// TIA Portal V20 export
DATA_BLOCK "HmiInterface"   // DB177
// stored: Access Published, MemoryReserve 100, Namespace Unit1.Em4
   VAR
      em : "LAF_typeEmInterface";
      cm : "Unit1.Em4.typeCmHmiInterface";
      sideTapeLoading : "LER_typeSequenceInterface";
      sideTapeAttachment : "LER_typeSequenceInterface";
      sideTapeFixStage : "LER_typeSequenceInterface";
      SideTapeIdleTime : "Unit1.Em4.typeSideTapeIdleTimeHmiInterface";
      sideTapeCuttingCount : "LER_typeAlarmCounterInterface";
      cmSideTapeSafetyPin : "LBC_typeDigitalSignalInterface";
      cmSideTapeJRDetect : "LBC_typeDigitalSignalInterface";
      cmSideTapeDiameter : "LBC_typeDigitalSignalInterface";
      cmSideTapeFixStageAxisX : "LBC_typeAxis64PosInterface";
      cmSideTapeFixStageAxisC : "LBC_typeAxis64PosInterface";
      cmSideTapeAttachmentAxisX : "LBC_typeAxis64PosInterface";
      cmSideTapeAttachmentAxisY : "LBC_typeAxis64PosInterface";
      cmSideTapeLoadingDownUp : "LBC_typeTwoWayActuatorInterface";
      cmSideTapeLoadingClampOpenClose : "LBC_typeTwoWayActuatorInterface";
      cmSideTapeCutterBwdFwd : "LBC_typeTwoWayActuatorInterface";
      cmSideTapeCutterClampBwdFwd : "LBC_typeTwoWayActuatorInterface";
      cmSideTapeTensionBwdFwd : "LBC_typeTwoWayActuatorInterface";
      cmSideTapeAttachmentLeftBwdFwd : "LBC_typeTwoWayActuatorInterface";
      cmSideTapeAttachmentRightBwdFwd : "LBC_typeTwoWayActuatorInterface";
      cmSideTapeAttachmentBtmBwdFwd : "LBC_typeTwoWayActuatorInterface";
      cmSideTapeFixStageClampOpenClose : "LBC_typeTwoWayActuatorInterface";
      cmSideTapeAttachment1TopVaccumOffOn : "LBC_typeTwoWayActuatorInterface";
      cmSideTapeAttachment1BtmVaccumOffOn : "LBC_typeTwoWayActuatorInterface";
      cmSideTapeAttachment2TopVaccumOffOn : "LBC_typeTwoWayActuatorInterface";
      cmSideTapeAttachment2BtmVaccumOffOn : "LBC_typeTwoWayActuatorInterface";
      cmQrHandyReader : "LER_typeDM8700Interface";
      "=====사용유무 확인필요=====" { ExternalAccessible := 'False'; ExternalVisible := 'False'; ExternalWritable := 'False'} : Bool;
      sequenceUnused : Array[0.._.U1EM4_NO_OF_SEQUENCE] of Bool;
      intCondition : "Unit1.Em4.typeIntConditionHmiInterface";
   END_VAR
BEGIN
   SideTapeIdleTime.processCount := T#5M;
   sideTapeCuttingCount.referenceDesignator := WSTRING#'Em4 Side Tape Cutting Count';
   sideTapeCuttingCount.ProcessValue.faultCount := 5000;
   sideTapeCuttingCount.SetValue.faultCount := 50000;
   cmSideTapeFixStageAxisC.configuration.setPositions[0]."name" := 'Wait [Tape1]';
   cmSideTapeFixStageAxisC.configuration.setPositions[1]."name" := 'Tape2';
   cmSideTapeFixStageAxisC.configuration.setPositions[2]."name" := 'Tape3';
   cmSideTapeFixStageAxisC.configuration.setPositions[3]."name" := 'Tape4';
   cmSideTapeAttachmentAxisX.configuration.setPositions[0]."name" := 'Wait';
   cmSideTapeAttachmentAxisX.configuration.setPositions[1]."name" := 'Right Tape Get';
   cmSideTapeAttachmentAxisX.configuration.setPositions[2]."name" := 'Left Tape Get';
   cmSideTapeAttachmentAxisX.configuration.setPositions[3]."name" := 'Tape1 Put';
   cmSideTapeAttachmentAxisX.configuration.setPositions[4]."name" := 'Tape2 Put';
   cmSideTapeAttachmentAxisX.configuration.setPositions[5]."name" := 'Tape3 Put';
   cmSideTapeAttachmentAxisX.configuration.setPositions[6]."name" := 'Tape4 Put';
   cmSideTapeAttachmentAxisX.configuration.setPositions[7]."name" := 'Remain Attachment Left';
   cmSideTapeAttachmentAxisX.configuration.setPositions[8]."name" := 'Remain Attachment Right';
   cmSideTapeAttachmentAxisX.configuration.setPositions[9]."name" := 'Tape Put Zone';
   cmSideTapeAttachmentAxisY.configuration.setPositions[0]."name" := 'Wait';
   cmSideTapeAttachmentAxisY.configuration.setPositions[1]."name" := 'Right Tape Get';
   cmSideTapeAttachmentAxisY.configuration.setPositions[2]."name" := 'Left Tape Get';
   cmSideTapeAttachmentAxisY.configuration.setPositions[3]."name" := 'Tape1 Put';
   cmSideTapeAttachmentAxisY.configuration.setPositions[4]."name" := 'Tape2 Put';
   cmSideTapeAttachmentAxisY.configuration.setPositions[5]."name" := 'Tape3 Put';
   cmSideTapeAttachmentAxisY.configuration.setPositions[6]."name" := 'Tape4 Put';
   cmSideTapeAttachmentAxisY.configuration.setPositions[7]."name" := 'Remain Attachment Left';
   cmSideTapeAttachmentAxisY.configuration.setPositions[8]."name" := 'Remain Attachment Right';
   cmSideTapeAttachmentAxisY.configuration.setPositions[9]."name" := 'No Interference Zone';
END_DATA_BLOCK
